Fanuc KAREL source: kt00368.KL

PROGRAM KT00368
%NOLOCKGROUP
VAR
I1:INTEGER
H2 : ARRAY[2] OF SHORT
OUT:BOOLEAN
BEGIN
I1=2
H2[1]=3
OUT=(I1<=H2[1])
END KT00368
